Staubli VAL3: getListItem.pgx

public program getListItem(string& x_sItem[], num x_nIndex)
  local trsf l_tTrsf
  local string l_sItem[6]
  local string l_sEvent
  local string l_sItem2[7]
begin
  //
  // define the item to show in the edit page Traj
  // customize an array and copy to x_sItem...
  //
  // see other traj as example
  // take it
  l_sEvent="coord  "
  l_tTrsf=pEditPoint.tData[x_nIndex].pPoint.trsf
  // show them
  l_sItem[0]=l_sItem2[0]=("coord  X > "+toString(".2",l_tTrsf.x))
  l_sItem[1]=l_sItem2[1]=("coord  Y > "+toString(".2",l_tTrsf.y))
  l_sItem[2]=l_sItem2[2]=("coord  Z > "+toString(".2",l_tTrsf.z))
  l_sItem[3]=l_sItem2[3]=("coord RX > "+toString(".2",l_tTrsf.rx))
  l_sItem[4]=l_sItem2[4]=("coord RY > "+toString(".2",l_tTrsf.ry))
  l_sItem[5]=l_sItem2[5]=("coord RZ > "+toString(".2",l_tTrsf.rz))
  // check the moveType
  if pEditPoint.tData[x_nIndex].tSuper.moveType==2
    // insert the circle POINT
    l_sItem2[6]="Point intermediate"
    call use:stringCopy(l_sItem2,x_sItem)
  else
    // look for intermediate point
    call use:stringCopy(l_sItem,x_sItem)
  endIf
end
